# EPICS autosave request: softGlueApp/Db/pixelTrigger_settings.req
$(P)$(Q)pixelTrigger.A
$(P)$(Q)pixelTrigger.B
$(P)$(Q)pixelTrigger.C
$(P)$(Q)pixelTrigger.SCAN
